{attribute 'qualified_only'}
{attribute 'strict'}
TYPE ABBLINKIN_RWS_API_VERSION :
(
	V1 := 0,
	V2 := 2
);
END_TYPE

(* stored: Version 1.1.0.1, ProductVersion 3.1.4024.12
   DUT ABBLINKIN_RWS_API_VERSION: Id {34efa19d-f9cb-43b8-bfe7-6b289ebee141} *)
